LIN {X 585.082, Y 308.882, Z 374.842, A -106.87, B 85.042, C -82.235, E1 0, E2 0, E3 0, E4 0}
LIN {X 583.182, Y 304.273, Z 375.273, A -106.87, B 85.042, C -82.235, E1 0, E2 0, E3 0, E4 0}
LIN {X 559.949, Y 314.912, Z 374.974, A -106.87, B 85.042, C -82.235, E1 0, E2 0, E3 0, E4 0}
LIN {X 559.915, Y 309.449, Z 375.429, A -106.87, B 85.042, C -82.235, E1 0, E2 0, E3 0, E4 0}
LIN {X 581.421, Y 299.6, Z 375.705, A -106.87, B 85.042, C -82.235, E1 0, E2 0, E3 0, E4 0}
LIN {X 579.153, Y 295.16, Z 376.131, A -106.87, B 85.042, C -82.235, E1 0, E2 0, E3 0, E4 0}
LIN {X 559.632, Y 304.099, Z 375.88, A -106.87, B 85.042, C -82.235, E1 0, E2 0, E3 0, E4 0}
LIN {X 559.38, Y 298.735, Z 376.332, A -106.87, B 85.042, C -82.235, E1 0, E2 0, E3 0, E4 0}
LIN {X 576.99, Y 290.671, Z 376.558, A -106.87, B 85.042, C -82.235, E1 0, E2 0, E3 0, E4 0}
LIN {X 575.354, Y 285.941, Z 376.992, A -106.87, B 85.042, C -82.235, E1 0, E2 0, E3 0, E4 0}
LIN {X 559.587, Y 293.162, Z 376.789, A -106.87, B 85.042, C -82.235, E1 0, E2 0, E3 0, E4 0}
LIN {X 559.173, Y 287.872, Z 377.239, A -106.87, B 85.042, C -82.235, E1 0, E2 0, E3 0, E4 0}
LIN {X 573.274, Y 281.414, Z 377.42, A -106.87, B 85.042, C -82.235, E1 0, E2 0, E3 0, E4 0}
LIN {X 571.532, Y 276.733, Z 377.852, A -106.87, B 85.042, C -82.235, E1 0, E2 0, E3 0, E4 0}
LIN {X 558.515, Y 282.694, Z 377.685, A -106.87, B 85.042, C -82.235, E1 0, E2 0, E3 0, E4 0}
LIN {X 558.353, Y 277.289, Z 378.138, A -106.87, B 85.042, C -82.235, E1 0, E2 0, E3 0, E4 0}
LIN {X 569.273, Y 272.288, Z 378.278, A -106.87, B 85.042, C -82.235, E1 0, E2 0, E3 0, E4 0}
LIN {X 567.396, Y 267.669, Z 378.709, A -106.87, B 85.042, C -82.235, E1 0, E2 0, E3 0, E4 0}
LIN {X 558.027, Y 271.959, Z 378.589, A -106.87, B 85.042, C -82.235, E1 0, E2 0, E3 0, E4 0}
LIN {X 557.888, Y 266.544, Z 379.042, A -106.87, B 85.042, C -82.235, E1 0, E2 0, E3 0, E4 0}
LIN {X 565.662, Y 262.983, Z 379.142, A -106.87, B 85.042, C -82.235, E1 0, E2 0, E3 0, E4 0}
LIN {X 578.568, Y 345.488, Z 371.967, A -106.87, B 85.042, C -82.235, E1 0, E2 0, E3 0, E4 0}
LIN {X 582.649, Y 344.212, Z 371.97, A -106.87, B 85.042, C -82.235, E1 0, E2 0, E3 0, E4 0}
LIN {X 596.406, Y 340.998, Z 371.891, A -106.87, B 85.042, C -82.235, E1 0, E2 0, E3 0, E4 0}
LIN {X 597.297, Y 339.764, Z 371.971, A -106.87, B 85.042, C -82.235, E1 0, E2 0, E3 0, E4 0}
LIN {X 598.296, Y 338.934, Z 372.015, A -106.87, B 85.042, C -82.235, E1 0, E2 0, E3 0, E4 0}
LIN {X 598.55, Y 338.454, Z 372.048, A -106.87, B 85.042, C -82.235, E1 0, E2 0, E3 0, E4 0}
LIN {X 598.433, Y 337.903, Z 372.097, A -106.87, B 85.042, C -82.235, E1 0, E2 0, E3 0, E4 0}
LIN {X 596.462, Y 334.102, Z 372.462, A -106.87, B 85.042, C -82.235, E1 0, E2 0, E3 0, E4 0}
LIN {X 596.42, Y 334.063, Z 372.466, A -106.87, B 85.042, C -82.235, E1 0, E2 0, E3 0, E4 0}
LIN {X 592.589, Y 324.81, Z 373.331, A -106.87, B 85.042, C -82.235, E1 0, E2 0, E3 0, E4 0}
LIN {X 591.868, Y 323.741, Z 373.438, A -106.87, B 85.042, C -82.235, E1 0, E2 0, E3 0, E4 0}
LIN {X 591.803, Y 323.313, Z 373.475, A -106.87, B 85.042, C -82.235, E1 0, E2 0, E3 0, E4 0}
LIN {X 591.302, Y 322.41, Z 373.563, A -106.87, B 85.042, C -82.235, E1 0, E2 0, E3 0, E4 0}
LIN {X 591.168, Y 321.833, Z 373.614, A -106.87, B 85.042, C -82.235, E1 0, E2 0, E3 0, E4 0}
LIN {X 590.595, Y 321.044, Z 373.694, A -106.87, B 85.042, C -82.235, E1 0, E2 0, E3 0, E4 0}
LIN {X 590.595, Y 321.03, Z 373.695, A -106.87, B 85.042, C -82.235, E1 0, E2 0, E3 0, E4 0}
LIN {X 589.218, Y 317.941, Z 373.986, A -106.87, B 85.042, C -82.235, E1 0, E2 0, E3 0, E4 0}
LIN {X 589.006, Y 316.394, Z 374.12, A -106.87, B 85.042, C -82.235, E1 0, E2 0, E3 0, E4 0}
LIN {X 587.25, Y 313.169, Z 374.432, A -106.87, B 85.042, C -82.235, E1 0, E2 0, E3 0, E4 0}
LIN {X 584.613, Y 307.292, Z 374.986, A -106.87, B 85.042, C -82.235, E1 0, E2 0, E3 0, E4 0}
LIN {X 584.337, Y 306.709, Z 375.041, A -106.87, B 85.042, C -82.235, E1 0, E2 0, E3 0, E4 0}
LIN {X 584.29, Y 306.409, Z 375.068, A -106.87, B 85.042, C -82.235, E1 0, E2 0, E3 0, E4 0}
LIN {X 582.357, Y 302.434, Z 375.446, A -106.87, B 85.042, C -82.235, E1 0, E2 0, E3 0, E4 0}
LIN {X 582.171, Y 301.694, Z 375.512, A -106.87, B 85.042, C -82.235, E1 0, E2 0, E3 0, E4 0}
LIN {X 577.158, Y 291.299, Z 376.501, A -106.87, B 85.042, C -82.235, E1 0, E2 0, E3 0, E4 0}
LIN {X 573.133, Y 281.193, Z 377.442, A -106.87, B 85.042, C -82.235, E1 0, E2 0, E3 0, E4 0}
LIN {X 572.429, Y 278.523, Z 377.681, A -106.87, B 85.042, C -82.235, E1 0, E2 0, E3 0, E4 0}
LIN {X 571.277, Y 276.036, Z 377.917, A -106.87, B 85.042, C -82.235, E1 0, E2 0, E3 0, E4 0}
LIN {X 570.712, Y 275.311, Z 377.991, A -106.87, B 85.042, C -82.235, E1 0, E2 0, E3 0, E4 0}
LIN {X 566.324, Y 265.712, Z 378.898, A -106.87, B 85.042, C -82.235, E1 0, E2 0, E3 0, E4 0}
LIN {X 565.184, Y 261.469, Z 379.279, A -106.87, B 85.042, C -82.235, E1 0, E2 0, E3 0, E4 0}
LIN {X 565.04, Y 260.787, Z 379.34, A -106.87, B 85.042, C -82.235, E1 0, E2 0, E3 0, E4 0}
LIN {X 565.02, Y 260.75, Z 379.343, A -106.87, B 85.042, C -82.235, E1 0, E2 0, E3 0, E4 0}
LIN {X 562.706, Y 261.377, Z 379.349, A -106.87, B 85.042, C -82.235, E1 0, E2 0, E3 0, E4 0}
LIN {X 562.668, Y 261.444, Z 379.345, A -106.87, B 85.042, C -82.235, E1 0, E2 0, E3 0, E4 0}
LIN {X 561.877, Y 261.598, Z 379.352, A -106.87, B 85.042, C -82.235, E1 0, E2 0, E3 0, E4 0}
LIN {X 561.428, Y 261.534, Z 379.369, A -106.87, B 85.042, C -82.235, E1 0, E2 0, E3 0, E4 0}
LIN {X 561.395, Y 261.421, Z 379.379, A -106.87, B 85.042, C -82.235, E1 0, E2 0, E3 0, E4 0}
LIN {X 559.991, Y 261.125, Z 379.439, A -106.87, B 85.042, C -82.235, E1 0, E2 0, E3 0, E4 0}
LIN {X 557.549, Y 261.883, Z 379.437, A -106.87, B 85.042, C -82.235, E1 0, E2 0, E3 0, E4 0}
LIN {X 556.928, Y 261.894, Z 379.452, A -106.87, B 85.042, C -82.235, E1 0, E2 0, E3 0, E4 0}
LIN {X 556.492, Y 262.398, Z 379.421, A -106.87, B 85.042, C -82.235, E1 0, E2 0, E3 0, E4 0}
LIN {X 556.2, Y 263.633, Z 379.326, A -106.87, B 85.042, C -82.235, E1 0, E2 0, E3 0, E4 0}
LIN {X 558.1, Y 267.281, Z 378.975, A -106.87, B 85.042, C -82.235, E1 0, E2 0, E3 0, E4 0}
LIN {X 558.046, Y 271.01, Z 378.667, A -106.87, B 85.042, C -82.235, E1 0, E2 0, E3 0, E4 0}
LIN {X 558.338, Y 275.035, Z 378.326, A -106.87, B 85.042, C -82.235, E1 0, E2 0, E3 0, E4 0}
LIN {X 559.974, Y 307.872, Z 375.558, A -106.87, B 85.042, C -82.235, E1 0, E2 0, E3 0, E4 0}
LIN {X 559.619, Y 312.754, Z 375.162, A -106.87, B 85.042, C -82.235, E1 0, E2 0, E3 0, E4 0}
LIN {X 560.017, Y 314.351, Z 375.019, A -106.87, B 85.042, C -82.235, E1 0, E2 0, E3 0, E4 0}
LIN {X 559.935, Y 315.38, Z 374.936, A -106.87, B 85.042, C -82.235, E1 0, E2 0, E3 0, E4 0}
LIN {X 559.9, Y 315.449, Z 374.931, A -106.87, B 85.042, C -82.235, E1 0, E2 0, E3 0, E4 0}
LIN {X 560.269, Y 328.893, Z 373.806, A -106.87, B 85.042, C -82.235, E1 0, E2 0, E3 0, E4 0}
LIN {X 560.192, Y 329.053, Z 373.794, A -106.87, B 85.042, C -82.235, E1 0, E2 0, E3 0, E4 0}
LIN {X 559.246, Y 334.358, Z 373.378, A -106.87, B 85.042, C -82.235, E1 0, E2 0, E3 0, E4 0}
LIN {X 559.418, Y 346.464, Z 372.368, A -106.87, B 85.042, C -82.235, E1 0, E2 0, E3 0, E4 0}
LIN {X 559.345, Y 346.722, Z 372.349, A -106.87, B 85.042, C -82.235, E1 0, E2 0, E3 0, E4 0}
LIN {X 559.388, Y 351.391, Z 371.96, A -106.87, B 85.042, C -82.235, E1 0, E2 0, E3 0, E4 0}
LIN {X 559.481, Y 352.298, Z 371.882, A -106.87, B 85.042, C -82.235, E1 0, E2 0, E3 0, E4 0}
LIN {X 560.102, Y 352.334, Z 371.864, A -106.87, B 85.042, C -82.235, E1 0, E2 0, E3 0, E4 0}
LIN {X 566.708, Y 350.942, Z 371.813, A -106.87, B 85.042, C -82.235, E1 0, E2 0, E3 0, E4 0}
LIN {X 567.658, Y 350.287, Z 371.843, A -106.87, B 85.042, C -82.235, E1 0, E2 0, E3 0, E4 0}
LIN {X 569.149, Y 346.884, Z 372.088, A -106.87, B 85.042, C -82.235, E1 0, E2 0, E3 0, E4 0}
LIN {X 569.452, Y 346.657, Z 372.1, A -106.87, B 85.042, C -82.235, E1 0, E2 0, E3 0, E4 0}
LIN {X 570.385, Y 346.464, Z 372.092, A -106.87, B 85.042, C -82.235, E1 0, E2 0, E3 0, E4 0}
LIN {X 570.628, Y 346.259, Z 372.103, A -106.87, B 85.042, C -82.235, E1 0, E2 0, E3 0, E4 0}
LIN {X 572.627, Y 345.578, Z 372.109, A -106.87, B 85.042, C -82.235, E1 0, E2 0, E3 0, E4 0}
LIN {X 577.685, Y 345.764, Z 371.967, A -106.87, B 85.042, C -82.235, E1 0, E2 0, E3 0, E4 0}
LIN {X 578.568, Y 345.488, Z 371.967, A -106.87, B 85.042, C -82.235, E1 0, E2 0, E3 0, E4 0}
PTP {X 576.895, Y 342.279, Z 426.279, A -106.87, B 85.042, C -82.235, E1 0, E2 0, E3 0, E4 0, S 'B010'}
PTP {A1 5, A2 -90, A3 100, A4 5, A5 -10, A6 -5, E1 0, E2 0, E3 0, E4 0} C_PTP
;ENDFOLD

END
